// Gets the lower bound index of the array of specified type.
FUNCTION F_GetUIntArrayLowerBound : T_Position // The lower bound index of the specified array.
VAR_IN_OUT
	arArray : ARRAY[*] OF UINT; // The array to query.
END_VAR

F_GetUIntArrayLowerBound := LOWER_BOUND(arArray, 1);

END_FUNCTION

(* stored: Version 1.1.0.1
   POU F_GetUIntArrayLowerBound: Id {55f02148-84cf-0e22-2bea-d55aaf062e6f}, SpecialFunc None *)
